{attribute 'GeneratedUsingTerminal: EK1100-0000-0018'}
{attribute addProperty BoxType "EK1100-0000-0018"}
{attribute addProperty Id "Beckhoff_EP3xxxEK1122Beckhoff_EP3xxxEK1122_EFCFC79A3196"}
{attribute addProperty CRC "2588853451"}
{attribute addProperty Size "3196"}
TYPE Beckhoff_EP3xxx_9A4EC4CB EXTENDS EK1100_1FC0878B :
STRUCT
	{attribute addProperty Name "Beckhoff_EP3xxxEK1122"}
	{attribute addProperty PreviousPort "Beckhoff EP3xxx : B"}
	Beckhoff_EP3xxxEK1122 : Beckhoff_EP3xxxEK1122_EFCFC79A;
END_STRUCT
END_TYPE

(* stored: Version 1.2.0.0, ProductVersion 3.1.4024.9
   DUT Beckhoff_EP3xxx_9A4EC4CB: Id {d3dc55f1-ab0e-4a31-8758-b2679a80a3b1} *)
